// SIMATIC S7-200 project (STEP 7-Micro/WIN), CPU 221 REL 01.10

ORGANIZATION_BLOCK 主程序:OB1
TITLE=
BEGIN
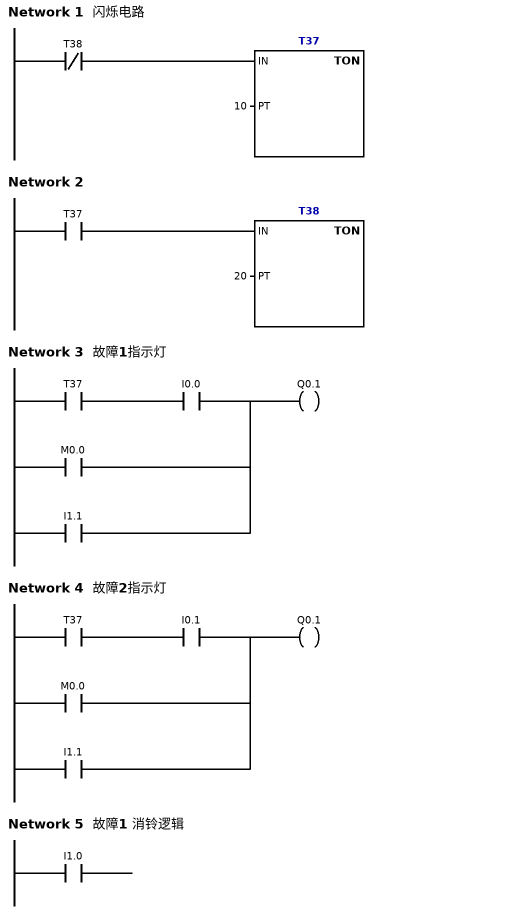
Network 1 // 闪烁电路
LDN    T38
TON    T37, 10
Network 2
LD     T37
TON    T38, 20
Network 3 // 故障1指示灯
LD     T37
A      I0.0
O      M0.0
O      I1.1
=      Q0.1
Network 4 // 故障2指示灯
LD     T37
A      I0.1
O      M0.0
O      I1.1
=      Q0.1
Network 5 // 故障1 消铃逻辑
// (network saved uncompiled; LAD cells follow)
// row 0: c0 -| |- I1.0
Network 6 // 故障2 消铃逻辑
Network 7 // 电铃
END_ORGANIZATION_BLOCK
